# EPICS StreamDevice protocol: camera-control/camera-controlApp/Db/cameracontrol.proto
http_headers = "Host: epicsss-axiscamera-01.cslab.esss.lu.se\r\nAuthorization: Basic cm9vdDplcGljcw==";

getParam {
    extrainput = ignore;
    out "GET /axis-cgi/param.cgi?action=list&group=\$1 HTTP/1.1\r\n"$http_headers"\r\n\r\n";
    in "%*/\$1=/%[^\r\n]";
}

setParam {
    extrainput = ignore;
    out "GET /axis-cgi/param.cgi?action=update&\$1=%s HTTP/1.1\r\n"$http_headers"\r\n\r\n";
}
